// TIA Portal project "az5" (V16)

(* hardware
DEVICE "S71500/ET200MP station_1"  S7-1500 station
   slot 0: "Rail_0"  Rack  6ES7 590-1***0-0AA0
   slot 1: "PLC_1"  CPU 1511C-1 PN  6ES7 511-1CK00-0AB0  V2.1
      slot 3: "CPU display_1"  6ES7591-1AA00-0AA0
      slot 32768: "PROFINET interface_1"  X1
         slot 32769: "Port_1"  X1 P1
         slot 32770: "Port_2"  X1 P2
*)

// ===== PLC "PLC_1"  CPU 1511C-1 PN =====

VAR_GLOBAL   // PLC tag table "Default tag table"
   "HIGH ALARM" AT %Q0.0 : Bool;
   "LOW ALARM" AT %Q0.1 : Bool;
   "HIGH ALARM(1)" AT %Q4.0 : Bool;
   "LOW ALARM(1)" AT %Q4.1 : Bool;
END_VAR

DATA_BLOCK "Data_block_1"   // DB2
{ S7_Optimized_Access := 'FALSE' }
VERSION : 0.1
   VAR
      D_SEL : Bool;
      I_SEL : Bool;
      P_SEL : Bool;
      GAIN : Real;
      TI : Time;
      TD : Time;
      SP_INT : Real;
      PV_IN : Real;
      MAN : Real;
      MAN_ON : Bool;
      LMN : Real;
      D_SEL_1 : Bool;
      I_SEL_1 : Bool;
      P_SEL_1 : Bool;
      GAIN_1 : Real;
      TI_1 : Time;
      TD_1 : Time;
      SP_INT_1 : Real;
      PV_IN_1 : Real;
      MAN_1 : Real;
      MAN_ON_1 : Bool;
      LMN_1 : Real;
   END_VAR
BEGIN
END_DATA_BLOCK

ORGANIZATION_BLOCK "Main"   // OB1, LAD, ProgramCycle
TITLE = "Main Program Sweep (Cycle)"
{ S7_Optimized_Access := 'TRUE' }
VERSION : 0.1
   VAR_INPUT
      Initial_Call : Bool;   // Initial call of this OB
      Remanence : Bool;   // =True, if remanent data are available
   END_VAR
BEGIN
END_ORGANIZATION_BLOCK

ORGANIZATION_BLOCK "Cyclic interrupt"   // OB30, LAD, CyclicInterrupt
{ S7_Optimized_Access := 'TRUE' }
VERSION : 0.1
   VAR_INPUT
      Initial_Call : Bool;   // Initial call of this OB
      Event_Count : Int;   // Events discarded
   END_VAR
BEGIN

REGION Network 1
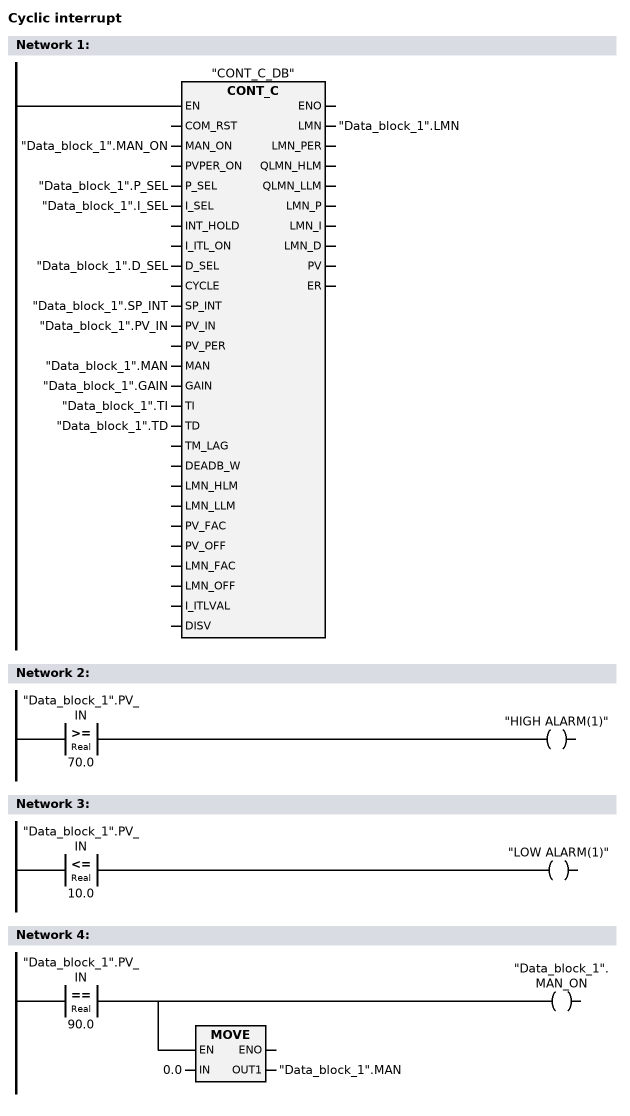
   "CONT_C_DB"(MAN_ON := "Data_block_1".MAN_ON,   // CONT_C
               P_SEL := "Data_block_1".P_SEL,
               I_SEL := "Data_block_1".I_SEL,
               D_SEL := "Data_block_1".D_SEL,
               SP_INT := "Data_block_1".SP_INT,
               PV_IN := "Data_block_1".PV_IN,
               MAN := "Data_block_1".MAN,
               GAIN := "Data_block_1".GAIN,
               TI := "Data_block_1".TI,
               TD := "Data_block_1".TD,
               LMN => "Data_block_1".LMN);
END_REGION

REGION Network 2
   RUNG wire#powerrail
      { S7_Templates := "SrcType := Real" } GE_Contact(in1 := "Data_block_1".PV_IN, in2 := 70.0)
      Coil( "HIGH ALARM(1)" )
   END_RUNG
   // the same network as SCL:
   "HIGH ALARM(1)" := "Data_block_1".PV_IN >= 70.0;
END_REGION

REGION Network 3
   RUNG wire#powerrail
      { S7_Templates := "SrcType := Real" } LE_Contact(in1 := "Data_block_1".PV_IN, in2 := 10.0)
      Coil( "LOW ALARM(1)" )
   END_RUNG
   // the same network as SCL:
   "LOW ALARM(1)" := "Data_block_1".PV_IN <= 10.0;
END_REGION

REGION Network 4
   RUNG wire#powerrail
      { S7_Templates := "SrcType := Real" } EQ_Contact(in1 := "Data_block_1".PV_IN, in2 := 90.0)
      wire#w1
      Coil( "Data_block_1".MAN_ON )
   END_RUNG
   RUNG wire#w1
      Move(in := 0.0, out1 => "Data_block_1".MAN)
   END_RUNG
   // the same network as SCL:
   "Data_block_1".MAN_ON := "Data_block_1".PV_IN = 90.0;
   IF "Data_block_1".MAN_ON THEN "Data_block_1".MAN := 0.0; END_IF;
END_REGION
END_ORGANIZATION_BLOCK